(* IEC 61131-3 sources: CodesysTest/export (part 4) *)

(* ---- FB_SolenoidValveManifold_UnitTests.st ---- *)
{attribute 'test' := 'multitest'}
{attribute 'testcasename':='Solenoid Valve Manifold Test'}
{attribute 'testcategory':='Solenoids'}
{attribute 'testcasetimeout':='15000'}
FUNCTION_BLOCK FB_SolenoidValveManifold_UnitTests EXTENDS CBM.EtrigA
VAR_INPUT
	xGetTestInfo : BOOL;
    diTestCaseIndex : DINT;
END_VAR
VAR_OUTPUT
    sTestCaseName : STRING;
	sTestCaseCategories : STRING;
    diTestCaseCount : DINT;
    diTestCaseTimeout : DINT;
    sInfo : STRING;
	eError : UnitTestErrors;
    sError : STRING;
    eFailureMode : TM.FAILUREMODE;
END_VAR
VAR
	valves : ARRAY[1..16] OF FB_DoubleSolenoidOpenCenterActuator(name := 'Unit Test Valve');
	testee : FB_SolenoidValveManifold(name := 'Unit Test Valve Manifold');
	testDWORD : DWORD;
END_VAR
SUPER^();
testee(ptrEIPOutputs := ADR(testDWORD));

{attribute 'hide'}
METHOD prvAbort : BOOL

SUPER^.prvAbort();

xAbortInProgress := FALSE;

{attribute 'hide'}
METHOD prvCyclicAction : BOOL

SUPER^.prvCyclicAction();
THIS^.diTestCaseCount := 6;

CASE diTestCaseIndex OF
    0: // Test Case #0
        IF THIS^.xGetTestInfo THEN
            THIS^.sTestCaseName := 'Step 1: Test All Solonoids Off';
            THIS^.sTestCaseCategories := 'Solenoids';
            THIS^.diTestCaseTimeout := 3000;
			xDone := TRUE;
		ELSE
			IF testDWORD = 0 THEN
				 xDone := TRUE;
			ELSE
				THIS^.sError := 'Solenoids not initalized off';
				xError := TRUE;
				eError := UnitTestErrors.Failure;
            	eFailureMode := TM.FAILUREMODE.AbortTestCase;
                iError := 1;
			END_IF
        END_IF
    1: // Test Case #1
        IF THIS^.xGetTestInfo THEN
            THIS^.sTestCaseName := 'Step 2: Extend Cylinder in Station 0';
            THIS^.sTestCaseCategories := 'Solenoids';
            THIS^.diTestCaseTimeout := 3000;
            xDone := TRUE;
		ELSE
			valves[1].Extend();
			testee();

			IF testDWORD = 1 THEN
				 xDone := TRUE;
			ELSE
				THIS^.sError := Standard.CONCAT('Incorrect bit set; value should be 1 was: ', TO_STRING(testDWORD));
				xError := TRUE;
				eError := UnitTestErrors.Failure;
            	eFailureMode := TM.FAILUREMODE.AbortTestCase;
                iError := 2;
			END_IF
       END_IF

	2:	//
		IF THIS^.xGetTestInfo THEN
            THIS^.sTestCaseName := 'Step 3: Retract Cylinder in Station 0';
            THIS^.sTestCaseCategories := 'Solenoids';
            THIS^.diTestCaseTimeout := 3000;
            xDone := TRUE;
		ELSE
			valves[1].Retract();
			testee();
			IF testDWORD = 2 THEN
				 xDone := TRUE;
			ELSE
				THIS^.sError := Standard.CONCAT('Incorrect bit set; value should be 2 was: ', TO_STRING(testDWORD));
				xError := TRUE;
				eError := UnitTestErrors.Failure;
            	eFailureMode := TM.FAILUREMODE.AbortTestCase;
                iError := 3;
			END_IF
       END_IF

   	3:	IF THIS^.xGetTestInfo THEN
            THIS^.sTestCaseName := 'Step 4: Extend Low Pressure Cylinder in Station 0';
            THIS^.sTestCaseCategories := 'Solenoids';
            THIS^.diTestCaseTimeout := 3000;
            xDone := TRUE;
		ELSE
			valves[1].ExtendLowPressure();
			testee();
			IF testDWORD = 3 THEN
				 xDone := TRUE;
			ELSE
				THIS^.sError := Standard.CONCAT('Incorrect bit set; value should be 2 was: ', TO_STRING(testDWORD));
				xError := TRUE;
				eError := UnitTestErrors.Failure;
            	eFailureMode := TM.FAILUREMODE.AbortTestCase;
                iError := 3;
			END_IF
       END_IF

	4: // Test Case #4
        IF THIS^.xGetTestInfo THEN
            THIS^.sTestCaseName := 'Step 5: Test Copy of Valve to 2nd position';
            THIS^.sTestCaseCategories := 'Solenoids';
            THIS^.diTestCaseTimeout := 3000;
			xDone := TRUE;
		ELSE
			testee.station[2] := valves[1];
			testee();
			IF testDWORD = 15 THEN
				 xDone := TRUE;
			ELSE
				THIS^.sError := Standard.CONCAT('Incorrect bits set; value should be 15 was: ', TO_STRING(testDWORD));
				xError := TRUE;
				eError := UnitTestErrors.Failure;
            	eFailureMode := TM.FAILUREMODE.AbortTestCase;
                iError := 1;
			END_IF
        END_IF

		5: // Test Case #5
        IF THIS^.xGetTestInfo THEN
            THIS^.sTestCaseName := 'Step 6: Exhaust Valves';
            THIS^.sTestCaseCategories := 'Solenoids';
            THIS^.diTestCaseTimeout := 3000;
			xDone := TRUE;
		ELSE
			valves[1].Exhaust();
			testee();
			IF testDWORD = 0 THEN
				 xDone := TRUE;
			ELSE
				THIS^.sError := Standard.CONCAT('Incorrect bits set; value should be 0 was: ', TO_STRING(testDWORD));
				xError := TRUE;
				eError := UnitTestErrors.Failure;
            	eFailureMode := TM.FAILUREMODE.AbortTestCase;
                iError := 1;
			END_IF
        END_IF

    ELSE
        IF THIS^.diTestCaseIndex < 0 THEN
            THIS^.diTestCaseCount := 6;
            xDone := TRUE;
        ELSE
            THIS^.sInfo := 'Invalid test case index';
            eError := UnitTestErrors.Failure;
			xError := TRUE;
        END_IF
END_CASE

{attribute 'hide'}
METHOD prvResetOutputs : BOOL

SUPER^.prvResetOutputs();

sTestCaseName := '';
sTestCaseCategories := '';
diTestCaseCount := 0;
diTestCaseTimeout := 0;
sInfo := '';
sError := '';
eFailureMode := TM.FAILUREMODE.AbortTestCase;

{attribute 'hide'}
METHOD prvStart : BOOL

SUPER^.prvStart();
testee.station[1] := valves[1];
testee.station[2] := valves[2];
testee.station[3] := valves[3];
testee.station[4] := valves[4];
testee.station[5] := valves[5];
testee.station[6] := valves[6];
testee.station[7] := valves[7];
testee.station[8] := valves[8];
testee.station[9] := valves[9];
testee.station[10] := valves[10];
testee.station[11] := valves[11];
testee.station[12] := valves[12];
testee.station[13] := valves[13];
testee.station[14] := valves[14];
testee.station[15] := valves[15];
testee.station[16] := valves[16];

{attribute 'test' := 'multitest'}
{attribute 'testcasename':='Solenoid Valve Manifold Test'}
{attribute 'testcategory':='Solenoids'}
{attribute 'testcasetimeout':='15000'}
FUNCTION_BLOCK FB_SolenoidValveManifold_UnitTests EXTENDS CBM.EtrigA
VAR_INPUT
	xGetTestInfo : BOOL;
    diTestCaseIndex : DINT;
END_VAR
VAR_OUTPUT
    sTestCaseName : STRING;
	sTestCaseCategories : STRING;
    diTestCaseCount : DINT;
    diTestCaseTimeout : DINT;
    sInfo : STRING;
	eError : UnitTestErrors;
    sError : STRING;
    eFailureMode : TM.FAILUREMODE;
END_VAR
VAR
	valves : ARRAY[1..16] OF FB_DoubleSolenoidOpenCenterActuator(name := 'Unit Test Valve');
	testee : FB_SolenoidValveManifold(name := 'Unit Test Valve Manifold');
	testDWORD : DWORD;
END_VAR
SUPER^();
testee(ptrEIPOutputs := ADR(testDWORD));

{attribute 'hide'}
METHOD prvAbort : BOOL

SUPER^.prvAbort();

xAbortInProgress := FALSE;

{attribute 'hide'}
METHOD prvCyclicAction : BOOL

SUPER^.prvCyclicAction();
THIS^.diTestCaseCount := 6;

CASE diTestCaseIndex OF
    0: // Test Case #0
        IF THIS^.xGetTestInfo THEN
            THIS^.sTestCaseName := 'Step 1: Test All Solonoids Off';
            THIS^.sTestCaseCategories := 'Solenoids';
            THIS^.diTestCaseTimeout := 3000;
			xDone := TRUE;
		ELSE
			IF testDWORD = 0 THEN
				 xDone := TRUE;
			ELSE
				THIS^.sError := 'Solenoids not initalized off';
				xError := TRUE;
				eError := UnitTestErrors.Failure;
            	eFailureMode := TM.FAILUREMODE.AbortTestCase;
                iError := 1;
			END_IF
        END_IF
    1: // Test Case #1
        IF THIS^.xGetTestInfo THEN
            THIS^.sTestCaseName := 'Step 2: Extend Cylinder in Station 0';
            THIS^.sTestCaseCategories := 'Solenoids';
            THIS^.diTestCaseTimeout := 3000;
            xDone := TRUE;
		ELSE
			valves[1].Extend();
			testee();

			IF testDWORD = 1 THEN
				 xDone := TRUE;
			ELSE
				THIS^.sError := Standard.CONCAT('Incorrect bit set; value should be 1 was: ', TO_STRING(testDWORD));
				xError := TRUE;
				eError := UnitTestErrors.Failure;
            	eFailureMode := TM.FAILUREMODE.AbortTestCase;
                iError := 2;
			END_IF
       END_IF

	2:	//
		IF THIS^.xGetTestInfo THEN
            THIS^.sTestCaseName := 'Step 3: Retract Cylinder in Station 0';
            THIS^.sTestCaseCategories := 'Solenoids';
            THIS^.diTestCaseTimeout := 3000;
            xDone := TRUE;
		ELSE
			valves[1].Retract();
			testee();
			IF testDWORD = 2 THEN
				 xDone := TRUE;
			ELSE
				THIS^.sError := Standard.CONCAT('Incorrect bit set; value should be 2 was: ', TO_STRING(testDWORD));
				xError := TRUE;
				eError := UnitTestErrors.Failure;
            	eFailureMode := TM.FAILUREMODE.AbortTestCase;
                iError := 3;
			END_IF
       END_IF

   	3:	IF THIS^.xGetTestInfo THEN
            THIS^.sTestCaseName := 'Step 4: Extend Low Pressure Cylinder in Station 0';
            THIS^.sTestCaseCategories := 'Solenoids';
            THIS^.diTestCaseTimeout := 3000;
            xDone := TRUE;
		ELSE
			valves[1].ExtendLowPressure();
			testee();
			IF testDWORD = 3 THEN
				 xDone := TRUE;
			ELSE
				THIS^.sError := Standard.CONCAT('Incorrect bit set; value should be 2 was: ', TO_STRING(testDWORD));
				xError := TRUE;
				eError := UnitTestErrors.Failure;
            	eFailureMode := TM.FAILUREMODE.AbortTestCase;
                iError := 3;
			END_IF
       END_IF

	4: // Test Case #4
        IF THIS^.xGetTestInfo THEN
            THIS^.sTestCaseName := 'Step 5: Test Copy of Valve to 2nd position';
            THIS^.sTestCaseCategories := 'Solenoids';
            THIS^.diTestCaseTimeout := 3000;
			xDone := TRUE;
		ELSE
			testee.station[2] := valves[1];
			testee();
			IF testDWORD = 15 THEN
				 xDone := TRUE;
			ELSE
				THIS^.sError := Standard.CONCAT('Incorrect bits set; value should be 15 was: ', TO_STRING(testDWORD));
				xError := TRUE;
				eError := UnitTestErrors.Failure;
            	eFailureMode := TM.FAILUREMODE.AbortTestCase;
                iError := 1;
			END_IF
        END_IF

		5: // Test Case #5
        IF THIS^.xGetTestInfo THEN
            THIS^.sTestCaseName := 'Step 6: Exhaust Valves';
            THIS^.sTestCaseCategories := 'Solenoids';
            THIS^.diTestCaseTimeout := 3000;
			xDone := TRUE;
		ELSE
			valves[1].Exhaust();
			testee();
			IF testDWORD = 0 THEN
				 xDone := TRUE;
			ELSE
				THIS^.sError := Standard.CONCAT('Incorrect bits set; value should be 0 was: ', TO_STRING(testDWORD));
				xError := TRUE;
				eError := UnitTestErrors.Failure;
            	eFailureMode := TM.FAILUREMODE.AbortTestCase;
                iError := 1;
			END_IF
        END_IF

    ELSE
        IF THIS^.diTestCaseIndex < 0 THEN
            THIS^.diTestCaseCount := 6;
            xDone := TRUE;
        ELSE
            THIS^.sInfo := 'Invalid test case index';
            eError := UnitTestErrors.Failure;
			xError := TRUE;
        END_IF
END_CASE

{attribute 'hide'}
METHOD prvResetOutputs : BOOL

SUPER^.prvResetOutputs();

sTestCaseName := '';
sTestCaseCategories := '';
diTestCaseCount := 0;
diTestCaseTimeout := 0;
sInfo := '';
sError := '';
eFailureMode := TM.FAILUREMODE.AbortTestCase;

{attribute 'hide'}
METHOD prvStart : BOOL

SUPER^.prvStart();
testee.station[1] := valves[1];
testee.station[2] := valves[2];
testee.station[3] := valves[3];
testee.station[4] := valves[4];
testee.station[5] := valves[5];
testee.station[6] := valves[6];
testee.station[7] := valves[7];
testee.station[8] := valves[8];
testee.station[9] := valves[9];
testee.station[10] := valves[10];
testee.station[11] := valves[11];
testee.station[12] := valves[12];
testee.station[13] := valves[13];
testee.station[14] := valves[14];
testee.station[15] := valves[15];
testee.station[16] := valves[16];

(* ---- FB_UN00_SharpMachine.st ---- *)
FUNCTION_BLOCK FINAL FB_UN00_SharpMachine EXTENDS FB_PackMLStates
VAR_INPUT
	faultActive : BOOL;
END_VAR
VAR_OUTPUT
	currentState : PACK_ML.State;
END_VAR
VAR
	automaticUnitMode	: PACK_ML.UnitMode; // Example unit mode for prodction
	simUnitMode			: PACK_ML.UnitMode; // Example unit mode for semi auto production
	manitUnitMode		: PACK_ML.UnitMode; // Example unit mode for setup
	unitModeManager		: PACK_ML.UnitModeManager; // Unit mode manager to switch between unitmodes
	currentUnitMode		: PACK_ML.IUnitMode;
	xInit				: BOOL := FALSE; // Flag for initialization
	xNextState : BOOL; // Next state from HMI
	sCurrentUnitModeName : STRING;
	baggerManager : EM01_BaggerHead_Manager(name := 'Bagger Head Manager');

	startMachine : BOOL;
	abortMachine : BOOL;
	resetONS : FB_ONS;
	resetMachine : BOOL;
	clearTimer : Standard.TON := (PT := T#3S);
	testResetSim : BOOL;
END_VAR

VAR_IN_OUT
	baggerHead : EM01_BaggerHead;
	discharge : EM02_Discharge;
	//baggerManager : EM01_Bagger_Manager;
END_VAR
// Setup of unit modes

IF NOT xInit THEN
	automaticUnitMode(		sName := UN00_Globals.sAutomatic,
							dwSupportedStates := PACK_ML.State.All - PACK_ML.State.Completing - PACK_ML.State.Complete - PACK_ML.State.Suspended - PACK_ML.State.Suspending - PACK_ML.State.UnSuspending,
							dwAllowsLeavingFromStates := PACK_ML.State.Stopped OR PACK_ML.State.Aborted OR PACK_ML.State.Idle,
							dwAllowsEnteringIntoStates := PACK_ML.State.Stopped OR PACK_ML.State.Aborted OR PACK_ML.State.Idle,
							eInitialState := PACK_ML.State.Stopped,
							xActive := TRUE);

	manitUnitMode(			sName := UN00_Globals.sMaintenance,
							dwSupportedStates := PACK_ML.State.All - PACK_ML.State.Completing - PACK_ML.State.Complete - PACK_ML.State.Holding - PACK_ML.State.Held - PACK_ML.State.UnHolding - PACK_ML.State.UnSuspending - PACK_ML.State.Suspended - PACK_ML.State.Suspending,
							dwAllowsLeavingFromStates := PACK_ML.State.Stopped OR PACK_ML.State.Aborted OR PACK_ML.State.Idle,
							dwAllowsEnteringIntoStates := PACK_ML.State.Stopped OR PACK_ML.State.Aborted OR PACK_ML.State.Idle,
							eInitialState := PACK_ML.State.Stopped,
							xActive := FALSE);

	// Register the unit modes
	unitModeManager.Register(automaticUnitMode);
	unitModeManager.Register(manitUnitMode);
	xInit := TRUE;
END_IF

currentUnitMode := unitModeManager.ActiveUnitMode;
sCurrentUnitModeName := currentUnitMode.Name;
currentState := currentUnitMode.CurrentState;
IF xNextState THEN
	currentUnitMode.Enter(currentUnitMode.NextState(currentUnitMode.CurrentState));
	xNextState := FALSE;
END_IF
baggerManager(
	modeManager := unitModeManager,
	baggerHead := baggerHead,
	discharge := discharge);

clearTimer();
resetONS(CLK := resetMachine);

IF testResetSim THEN
	UN00_Globals.simFaults.FB_Init(TRUE,TRUE);
END_IF

CASE unitModeManager.ActiveUnitMode.CurrentState OF

	PACK_ML.State.Stopped: 		IF resetONS.OSR OR _clearingDone THEN
									currentUnitMode.Reset();
								END_IF
								_clearingDone := FALSE;

	PACK_ML.State.Aborted:		IF resetONS.OSR THEN
									GlobalObjects.CollectionOfActiveFaults.AckAll();
									currentUnitMode.Clear();
								END_IF

	PACK_ML.State.Idle:			currentUnitMode.Start();

	PACK_ML.State.Held:			currentUnitMode.Unhold();
	//PACK_ML.State.Complete:
	PACK_ML.State.Resetting:	IF BaggerManager.ResettingDone THEN
									currentUnitMode.ActingStateCompleted();
								END_IF

	PACK_ML.State.Clearing :	clearTimer.IN := TRUE;
								IF BaggerManager.ClearingDone AND NOT faultActive THEN
									currentUnitMode.ActingStateCompleted();
									clearTimer.IN := FALSE;
									_clearingDone := TRUE;
								ELSIF clearTimer.Q THEN
									currentUnitMode.Abort();
									clearTimer.IN := FALSE;
								END_IF

	PACK_ML.State.Starting :	IF BaggerManager.StartingDone THEN
									currentUnitMode.ActingStateCompleted();
								END_IF

	//PACK_ML.State.Execute :
	PACK_ML.State.Holding :		IF BaggerManager.HoldingDone THEN
									currentUnitMode.ActingStateCompleted();
								END_IF
	//PACK_ML.State.UnHolding :
	//PACK_ML.State.Completing :
	PACK_ML.State.Aborting :	IF BaggerManager.AbortingDone THEN
									currentUnitMode.ActingStateCompleted();
								END_IF

	PACK_ML.State.Stopping:
								IF BaggerManager.StoppingDone THEN
									currentUnitMode.ActingStateCompleted();
								END_IF

END_CASE

IF (faultActive AND unitModeManager.ActiveUnitMode.CurrentState <> PACK_ML.State.Clearing) OR abortMachine THEN
	currentUnitMode.Abort();
	abortMachine := FALSE;
END_IF

startMachine := FALSE;

(* ---- FB_VacuumGenerator.st ---- *)
FUNCTION_BLOCK FB_VacuumGenerator EXTENDS FB_SolenoidValve
VAR_INPUT
END_VAR
VAR_OUTPUT
END_VAR
VAR
END_VAR

METHOD GeneratorsOn
VAR_INPUT
END_VAR

THIS^.solenoid0 := TRUE;
THIS^.solenoid1 := FALSE;

METHOD GeneratorsOff
VAR_INPUT
END_VAR

THIS^.solenoid0 := FALSE;
THIS^.solenoid1 := FALSE;

FUNCTION_BLOCK FB_VacuumGenerator EXTENDS FB_SolenoidValve
VAR_INPUT
END_VAR
VAR_OUTPUT
END_VAR
VAR
END_VAR

METHOD GeneratorsOn
VAR_INPUT
END_VAR

THIS^.solenoid0 := TRUE;
THIS^.solenoid1 := FALSE;

METHOD GeneratorsOff
VAR_INPUT
END_VAR

THIS^.solenoid0 := FALSE;
THIS^.solenoid1 := FALSE;

(* ---- Devices.st ---- *)
PROGRAM Devices
VAR

END_VAR
VAR_IN_OUT

END_VAR

VAR_OUTPUT

	IOMaster : FB_MurrMaster(name := 'IO Master') := 	(ptrEIPInputs := ADR(IOEIPInputs),
														 ptrEIPOutputs := ADR(IOEIPOutputs));

	pressureBarSolenoidValve : FB_DoubleSolenoidOpenCenterActuator(name := 'Pressure Bar SV');
	sealBarSolenoidValve : FB_SingleSolenoidNormallyRetractedActuator(name := 'Seal Bar SV');
	HPA_LPA_SolenoidValve : FB_DoubleSolenoidClosedCenterActuator(name := 'HPA/LPA SV');
	loadPlateSolenoidValve : FB_DoubleSolenoidOpenCenterActuator(name := 'Load Plate SV');
	bagOpenFingersSolenoidValve : FB_DoubleSolenoidOpenCenterActuator(name := 'BOF SV');
	printHeadSolenoidValve : FB_SingleSolenoidNormallyRetractedActuator(name := 'Print Head SV');
	vacuumSolenoidValve : FB_VacuumGenerator(name := 'Vacuum SV');
	sealFlattenersVertAxisSolenoidValve : FB_DoubleSolenoidOpenCenterActuator(name := 'Seal Flattener Vert SV');
	loadShelfSolenoidValve : FB_DoubleSolenoidOpenCenterActuator(name := 'Load Shelf SV');
	blankSolenoidValve : FB_SolenoidValve(name := 'Blank SV');
	i : UINT;

	valveManifold : FB_SolenoidValveManifold(name := 'Valve Manifold') := (ptrEIPOutputs := ADR(Valve_Manifold_Outputs));

END_VAR

// Valve manifold station selection
FOR i := 1 TO Globals.MAX_VALVE_MANIFOLD_STATIONS DO
	CASE HMI.data.stationValveSelection[i] OF

		ValveSelection.PressureBar : 						valveManifold.station[i] := pressureBarSolenoidValve;

		ValveSelection.SealBar : 							valveManifold.station[i] := sealBarSolenoidValve;

		ValveSelection.HPA_LPA : 							valveManifold.station[i] := HPA_LPA_SolenoidValve;

		ValveSelection.LoadPlate : 							valveManifold.station[i] := loadPlateSolenoidValve;

		ValveSelection.BagOpenFingers : 					valveManifold.station[i] := bagOpenFingersSolenoidValve;

		ValveSelection.PrintHead : 							valveManifold.station[i] := printHeadSolenoidValve;

		ValveSelection.Vacuum : 							valveManifold.station[i] := vacuumSolenoidValve;

		ValveSelection.SealFlattenersVerticalAxis : 		valveManifold.station[i] := sealFlattenersVertAxisSolenoidValve;

		ValveSelection.LoadShelf : 							valveManifold.station[i] := loadShelfSolenoidValve;

		ValveSelection.Blank : 								valveManifold.station[i] := blankSolenoidValve;

	ELSE
		valveManifold.station[i] := blankSolenoidValve;
	END_CASE
END_FOR

// Run all configured valves and then the manifold
pressureBarSolenoidValve();
sealBarSolenoidValve();
HPA_LPA_SolenoidValve();
loadPlateSolenoidValve();
bagOpenFingersSolenoidValve();
printHeadSolenoidValve();
vacuumSolenoidValve();
sealFlattenersVertAxisSolenoidValve();
loadShelfSolenoidValve();
blankSolenoidValve();
valveManifold();

IOMaster();

(* ---- Main_PRG.st ---- *)
PROGRAM Main_PRG
VAR

	firstScanDone : BOOL;
	UN00_Pro18Machine : FB_UN00_SharpMachine(name := 'UN00 - Sharp Pro-18');
	EM01_Pro18BaggerHead : EM01_BaggerHead(name := 'EM01 - Pro 18 Bagger Head');
	EM02_Pro18Discharge : EM02_Discharge(name := 'EM02 - Pro 18 Discharge');
	activeBaggerHead : REFERENCE TO EM01_BaggerHead;
	machineComponents : EM01_Bagger_Control_Modules();

	activeBagOpenFingers : IBagOpenFingers := machineComponents.standardBagOpenFingersWithSensors;
	activeSealFlatteners : ISealFlatteners;
	activePressureBar : IPressureBar;
	activeSealer : ISealer;
	activePrinter : IPrinter;
	activeBagDelivery : IBagDelivery;
	activeRetractingLoadPlate : IRetractingLoadPlate;
	activeExitConveyor : IExitConveyor;
	activeVacuumBagOpen : IVacuumBagOpen;

	powerUpPassthroughMotor : Sharp_Motion.MC_Power;
	powerUpMSFHorizMotor : Sharp_Motion.MC_Power;
	powerUpBagDeliveryMotor : Sharp_Motion.MC_Power;

END_VAR
{IF defined (IsSimulationMode)}
	HMI.data.simulateAllIO := TRUE;
{END_IF}

Devices();
machineComponents();

powerUpPassthroughMotor(Enable := TRUE, Axis := machineComponents.passthroughMotor);
powerUpPassthroughMotor.DriveStart := TRUE;
powerUpPassthroughMotor.RegulatorOn := TRUE;

powerUpMSFHorizMotor(Enable := TRUE, Axis := machineComponents.msfHorizontalMotor);
powerUpMSFHorizMotor.DriveStart := TRUE;
powerUpMSFHorizMotor.RegulatorOn := TRUE;

powerUpBagDeliveryMotor(Enable := TRUE, Axis := machineComponents.bagDeliveryFrontMotor);
powerUpBagDeliveryMotor.DriveStart := TRUE;
powerUpBagDeliveryMotor.RegulatorOn := TRUE;

CASE HMI.data.bofSelection OF
	BagOpenFingersSelection.NotInstalled:
															activeBagOpenFingers := machineComponents.standardBagOpenFingersWithSensors;
															activeBagOpenFingers.OptionInstalled := FALSE;

	BagOpenFingersSelection.PneumaticWithBagOpenSensors: 	activeBagOpenFingers := machineComponents.standardBagOpenFingersWithSensors;
															activeBagOpenFingers.OptionInstalled := TRUE;
															activeBagOpenFingers.OptionEnabled := HMI.data.bofEnable;
END_CASE

CASE HMI.data.sealFlattenersSelection OF
	SealFlattenerSelection.NotInstalled:					activeSealFlatteners := machineComponents.motorizedSealFlatteners;
															activeSealFlatteners.OptionInstalled := FALSE;

	SealFlattenerSelection.MotorizedSealFlatteners:			activeSealFlatteners := machineComponents.motorizedSealFlatteners;
															activeSealFlatteners.OptionInstalled := TRUE;
															activeSealFlatteners.OptionEnabled := HMI.data.sealFlattenersEnable;
END_CASE

CASE HMI.data.printerSelection OF
	LabelPrinterSelection.NotInstalled:						activePrinter := machineComponents.labelPrinter;
															activePrinter.OptionInstalled := FALSE;

	LabelPrinterSelection.ZebraPrinter:						activePrinter := machineComponents.labelPrinter;
															activePrinter.OptionInstalled := TRUE;
															activePrinter.OptionEnabled := HMI.data.printerEnable;
END_CASE

EM01_Pro18BaggerHead(
	bagOpenFingers:= activeBagOpenFingers,
	sealFlatteners:= activeSealFlatteners,
	sealer:= machineComponents.standardSealBar,
	pressureBar:= machineComponents.pneumaticPressureBar,
	printer:= activePrinter,
	bagDelivery:= machineComponents.bagDelivery,
	vacuumBagOpen:= machineComponents.vacuumCups,
	bagOpenAssistEnabled:= HMI.data.bagOpenAssistEnable,
	bagOpenSensorEnabled:= HMI.data.bagOpenSensorEnable,
	separateBeforeSealEnabled:= HMI.data.separateBeforeSeal,
	bagOpenRetrySetting:= HMI.data.bagOpenRetrySetting,
	vacuumDwell := TO_TIME(HMI.data.vacuumDwell * 1000),
	baggerCycleActive=> ,
	bagOpenRetryCount=> HMI.data.bagOpenRetryCount);

activeBaggerHead REF= EM01_Pro18BaggerHead;
UN00_Pro18Machine(
	faultActive := HMI.data.faultActive,
	baggerHead := activeBaggerHead,
	discharge := EM02_Pro18Discharge);

Globals.SystemLog();

IF NOT firstScanDone THEN
	GlobalObjects.CollectionOfInitialzable.InitializeAll();
	GlobalObjects.CollectionOfLoggable.RegisterAll(internalLogger := Globals.SystemLog);
	GlobalObjects.CollectionOfFaults.FaultUpdateForHMI();
	firstScanDone := TRUE;
END_IF

HMI.data.faultActive := GlobalObjects.CollectionOfActiveFaults.faultActive;
IF HMI.data.ackAllFaults THEN
	GlobalObjects.CollectionOfActiveFaults.AckAll();
	HMI.data.ackAllFaults := FALSE;
END_IF

IF HMI.data.initiateCycle THEN
	IF UN00_Pro18Machine.currentState = PACK_ML.State.Execute THEN
		activeBaggerHead.StartCycle();
	END_IF
	HMI.data.initiateCycle := FALSE;
END_IF

IF firstScanDone THEN
	GlobalObjects.CollectionOfExecutable.ExecuteAll();
END_IF

(* ---- PLC_PRG.st ---- *)
PROGRAM PLC_PRG
VAR

	firstScanDone : BOOL;
	UN00_Pro18Machine : FB_UN00_SharpMachine(name := 'UN00 - Sharp Pro-18');
	EM01_Pro18BaggerHead : EM01_BaggerHead(name := 'EM01 - Pro 18 Bagger Head');
	EM02_Pro18Discharge : EM02_Discharge(name := 'EM02 - Pro 18 Discharge');
	activeBaggerHead : REFERENCE TO EM01_BaggerHead;
	machineComponents : EM01_Bagger_Control_Modules();

	activeBagOpenFingers : IBagOpenFingers := machineComponents.standardBagOpenFingersWithSensors;
	activeSealFlatteners : ISealFlatteners;
	activePressureBar : IPressureBar;
	activeSealer : ISealer;
	activePrinter : IPrinter;
	activeBagDelivery : IBagDelivery;
	activeRetractingLoadPlate : IRetractingLoadPlate;
	activeExitConveyor : IExitConveyor;
	activeVacuumBagOpen : IVacuumBagOpen;

	powerUpPassthroughMotor : Sharp_Motion.MC_Power;
	powerUpMSFHorizMotor : Sharp_Motion.MC_Power;
	powerUpBagDeliveryMotor : Sharp_Motion.MC_Power;

END_VAR
{IF defined (IsSimulationMode)}
	HMI.data.simulateAllIO := TRUE;
{END_IF}

Devices();
machineComponents();

powerUpPassthroughMotor(Enable := TRUE, Axis := machineComponents.passthroughMotor);
powerUpPassthroughMotor.DriveStart := TRUE;
powerUpPassthroughMotor.RegulatorOn := TRUE;

powerUpMSFHorizMotor(Enable := TRUE, Axis := machineComponents.msfHorizontalMotor);
powerUpMSFHorizMotor.DriveStart := TRUE;
powerUpMSFHorizMotor.RegulatorOn := TRUE;

powerUpBagDeliveryMotor(Enable := TRUE, Axis := machineComponents.bagDeliveryFrontMotor);
powerUpBagDeliveryMotor.DriveStart := TRUE;
powerUpBagDeliveryMotor.RegulatorOn := TRUE;

CASE HMI.data.bofSelection OF
	BagOpenFingersSelection.NotInstalled:
															activeBagOpenFingers := machineComponents.standardBagOpenFingersWithSensors;
															activeBagOpenFingers.OptionInstalled := FALSE;

	BagOpenFingersSelection.PneumaticWithBagOpenSensors: 	activeBagOpenFingers := machineComponents.standardBagOpenFingersWithSensors;
															activeBagOpenFingers.OptionInstalled := TRUE;
															activeBagOpenFingers.OptionEnabled := HMI.data.bofEnable;
END_CASE

CASE HMI.data.sealFlattenersSelection OF
	SealFlattenerSelection.NotInstalled:					activeSealFlatteners := machineComponents.motorizedSealFlatteners;
															activeSealFlatteners.OptionInstalled := FALSE;

	SealFlattenerSelection.MotorizedSealFlatteners:			activeSealFlatteners := machineComponents.motorizedSealFlatteners;
															activeSealFlatteners.OptionInstalled := TRUE;
															activeSealFlatteners.OptionEnabled := HMI.data.sealFlattenersEnable;
END_CASE

CASE HMI.data.printerSelection OF
	LabelPrinterSelection.NotInstalled:						activePrinter := machineComponents.labelPrinter;
															activePrinter.OptionInstalled := FALSE;

	LabelPrinterSelection.ZebraPrinter:						activePrinter := machineComponents.labelPrinter;
															activePrinter.OptionInstalled := TRUE;
															activePrinter.OptionEnabled := HMI.data.printerEnable;
END_CASE

EM01_Pro18BaggerHead(
	bagOpenFingers:= activeBagOpenFingers,
	sealFlatteners:= activeSealFlatteners,
	sealer:= machineComponents.standardSealBar,
	pressureBar:= machineComponents.pneumaticPressureBar,
	printer:= activePrinter,
	bagDelivery:= machineComponents.bagDelivery,
	vacuumBagOpen:= machineComponents.vacuumCups,
	bagOpenAssistEnabled:= HMI.data.bagOpenAssistEnable,
	bagOpenSensorEnabled:= HMI.data.bagOpenSensorEnable,
	separateBeforeSealEnabled:= HMI.data.separateBeforeSeal,
	bagOpenRetrySetting:= HMI.data.bagOpenRetrySetting,
	vacuumDwell := TO_TIME(HMI.data.vacuumDwell * 1000),
	baggerCycleActive=> ,
	bagOpenRetryCount=> HMI.data.bagOpenRetryCount);

activeBaggerHead REF= EM01_Pro18BaggerHead;
UN00_Pro18Machine(
	faultActive := HMI.data.faultActive,
	baggerHead := activeBaggerHead,
	discharge := EM02_Pro18Discharge);

Globals.SystemLog();

IF NOT firstScanDone THEN
	GlobalObjects.CollectionOfInitialzable.InitializeAll();
	GlobalObjects.CollectionOfLoggable.RegisterAll(internalLogger := Globals.SystemLog);
	GlobalObjects.CollectionOfFaults.FaultUpdateForHMI();
	firstScanDone := TRUE;
END_IF

HMI.data.faultActive := GlobalObjects.CollectionOfActiveFaults.faultActive;
IF HMI.data.ackAllFaults THEN
	GlobalObjects.CollectionOfActiveFaults.AckAll();
	HMI.data.ackAllFaults := FALSE;
END_IF

IF HMI.data.initiateCycle THEN
	IF UN00_Pro18Machine.currentState = PACK_ML.State.Execute THEN
		activeBaggerHead.StartCycle();
	END_IF
	HMI.data.initiateCycle := FALSE;
END_IF

IF firstScanDone THEN
	GlobalObjects.CollectionOfExecutable.ExecuteAll();
END_IF

PROGRAM PLC_PRG
VAR
	firstScan : BOOL; //First Scan Bit
	firstScanDone : BOOL; //First Scan Bit
	SystemLog : FB_InternalLogger;
END_VAR

SystemLog();

IF NOT firstScanDone THEN
	GlobalObjects.CollectionOfInitialzable.InitializeAll();
	GlobalObjects.CollectionOfLoggable.RegisterAll(internalLogger := SystemLog);
	GlobalObjects.CollectionOfFaults.FaultUpdateForHMI();
	firstScanDone := TRUE;
END_IF

PROGRAM PLC_PRG
VAR

	firstScanDone : BOOL;
	UN00_Pro18Machine : FB_UN00_SharpMachine(name := 'UN00 - Sharp Pro-18');
	EM01_Pro18BaggerHead : EM01_BaggerHead(name := 'EM01 - Pro 18 Bagger Head');
	EM02_Pro18Discharge : EM02_Discharge(name := 'EM02 - Pro 18 Discharge');
	activeBaggerHead : REFERENCE TO EM01_BaggerHead;
	machineComponents : EM01_Bagger_Control_Modules();

	activeBagOpenFingers : IBagOpenFingers := machineComponents.standardBagOpenFingersWithSensors;
	activeSealFlatteners : ISealFlatteners;
	activePressureBar : IPressureBar;
	activeSealer : ISealer;
	activePrinter : IPrinter;
	activeBagDelivery : IBagDelivery;
	activeRetractingLoadPlate : IRetractingLoadPlate;
	activeExitConveyor : IExitConveyor;
	activeVacuumBagOpen : IVacuumBagOpen;

	powerUpPassthroughMotor : Sharp_Motion.MC_Power;
	powerUpMSFHorizMotor : Sharp_Motion.MC_Power;
	powerUpBagDeliveryMotor : Sharp_Motion.MC_Power;

END_VAR
{IF defined (IsSimulationMode)}
	HMI.data.simulateAllIO := TRUE;
{END_IF}

Devices();
machineComponents();

powerUpPassthroughMotor(Enable := TRUE, Axis := machineComponents.passthroughMotor);
powerUpPassthroughMotor.DriveStart := TRUE;
powerUpPassthroughMotor.RegulatorOn := TRUE;

powerUpMSFHorizMotor(Enable := TRUE, Axis := machineComponents.msfHorizontalMotor);
powerUpMSFHorizMotor.DriveStart := TRUE;
powerUpMSFHorizMotor.RegulatorOn := TRUE;

powerUpBagDeliveryMotor(Enable := TRUE, Axis := machineComponents.bagDeliveryFrontMotor);
powerUpBagDeliveryMotor.DriveStart := TRUE;
powerUpBagDeliveryMotor.RegulatorOn := TRUE;

CASE HMI.data.bofSelection OF
	BagOpenFingersSelection.NotInstalled:
															activeBagOpenFingers := machineComponents.standardBagOpenFingersWithSensors;
															activeBagOpenFingers.OptionInstalled := FALSE;

	BagOpenFingersSelection.PneumaticWithBagOpenSensors: 	activeBagOpenFingers := machineComponents.standardBagOpenFingersWithSensors;
															activeBagOpenFingers.OptionInstalled := TRUE;
															activeBagOpenFingers.OptionEnabled := HMI.data.bofEnable;
END_CASE

CASE HMI.data.sealFlattenersSelection OF
	SealFlattenerSelection.NotInstalled:					activeSealFlatteners := machineComponents.motorizedSealFlatteners;
															activeSealFlatteners.OptionInstalled := FALSE;

	SealFlattenerSelection.MotorizedSealFlatteners:			activeSealFlatteners := machineComponents.motorizedSealFlatteners;
															activeSealFlatteners.OptionInstalled := TRUE;
															activeSealFlatteners.OptionEnabled := HMI.data.sealFlattenersEnable;
END_CASE

CASE HMI.data.printerSelection OF
	LabelPrinterSelection.NotInstalled:						activePrinter := machineComponents.labelPrinter;
															activePrinter.OptionInstalled := FALSE;

	LabelPrinterSelection.ZebraPrinter:						activePrinter := machineComponents.labelPrinter;
															activePrinter.OptionInstalled := TRUE;
															activePrinter.OptionEnabled := HMI.data.printerEnable;
END_CASE

EM01_Pro18BaggerHead(
	bagOpenFingers:= activeBagOpenFingers,
	sealFlatteners:= activeSealFlatteners,
	sealer:= machineComponents.standardSealBar,
	pressureBar:= machineComponents.pneumaticPressureBar,
	printer:= activePrinter,
	bagDelivery:= machineComponents.bagDelivery,
	vacuumBagOpen:= machineComponents.vacuumCups,
	bagOpenAssistEnabled:= HMI.data.bagOpenAssistEnable,
	bagOpenSensorEnabled:= HMI.data.bagOpenSensorEnable,
	separateBeforeSealEnabled:= HMI.data.separateBeforeSeal,
	bagOpenRetrySetting:= HMI.data.bagOpenRetrySetting,
	vacuumDwell := TO_TIME(HMI.data.vacuumDwell * 1000),
	baggerCycleActive=> ,
	bagOpenRetryCount=> HMI.data.bagOpenRetryCount);

activeBaggerHead REF= EM01_Pro18BaggerHead;
UN00_Pro18Machine(
	faultActive := HMI.data.faultActive,
	baggerHead := activeBaggerHead,
	discharge := EM02_Pro18Discharge);

Globals.SystemLog();

IF NOT firstScanDone THEN
	GlobalObjects.CollectionOfInitialzable.InitializeAll();
	GlobalObjects.CollectionOfLoggable.RegisterAll(internalLogger := Globals.SystemLog);
	GlobalObjects.CollectionOfFaults.FaultUpdateForHMI();
	firstScanDone := TRUE;
END_IF

HMI.data.faultActive := GlobalObjects.CollectionOfActiveFaults.faultActive;
IF HMI.data.ackAllFaults THEN
	GlobalObjects.CollectionOfActiveFaults.AckAll();
	HMI.data.ackAllFaults := FALSE;
END_IF

IF HMI.data.initiateCycle THEN
	IF UN00_Pro18Machine.currentState = PACK_ML.State.Execute THEN
		activeBaggerHead.StartCycle();
	END_IF
	HMI.data.initiateCycle := FALSE;
END_IF

IF firstScanDone THEN
	GlobalObjects.CollectionOfExecutable.ExecuteAll();
END_IF

PROGRAM PLC_PRG
VAR
	firstScan : BOOL; //First Scan Bit
	firstScanDone : BOOL; //First Scan Bit
	SystemLog : FB_InternalLogger;
END_VAR

SystemLog();

IF NOT firstScanDone THEN
	GlobalObjects.CollectionOfInitialzable.InitializeAll();
	GlobalObjects.CollectionOfLoggable.RegisterAll(internalLogger := SystemLog);
	GlobalObjects.CollectionOfFaults.FaultUpdateForHMI();
	firstScanDone := TRUE;
END_IF
